FUNCTION_BLOCK CyclicComponent_Mockup EXTENDS CyclicComponent IMPLEMENTS I_Resettable
VAR
	_WasCalled : BOOL;
END_VAR

METHOD CyclicLogic
_WasCalled := TRUE;
END_METHOD

METHOD Reset
END_METHOD

PROPERTY WasCalled : BOOL
GET
WasCalled := _WasCalled;
END_GET
END_PROPERTY

END_FUNCTION_BLOCK

(* stored: Version 1.1.0.1, ProductVersion 3.1.4026.18
   POU CyclicComponent_Mockup: Id {fe8d9105-ae63-474d-b6c3-ab28ccdb43db}, SpecialFunc None
   Method CyclicLogic: Id {e3e4c74d-7c34-4a9f-a2c5-a4aa377bdbd2}
   Method Reset: Id {e08bd1d7-21e9-406e-8f02-94a155a8ca5e}
   Property WasCalled: Id {f3896350-1690-4687-b6a2-3ee3e321c2fd}
   Get Get: Id {658661b0-20e5-41b3-a498-b4314d4192d4} *)
